SUBAPPLICATION AX_SPLIT_TO_2x_AX_TP (* 1 AX-Eingang gesplittet auf 2 unabhaengig retriggerbare Pulstimer (AX_TP), je eigene Pulsdauer (TQ1/TQ2) und eigener AX-Ausgang (Q1/Q2). Generisch, hardwareunabhaengig. *)
  (* Standard: 61499-2 *)
  (* Version 1.0, 2026-09-09, Franz Höpfinger, Meisterschulen am Ostbahnhof, Ausgelagert aus Uebung_020j2_AX_sub zur Wiederverwendung. *)
  PACKAGE MyLib::sys;
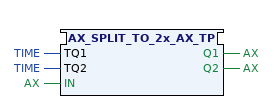
  VAR_INPUT
    TQ1 : TIME;
    TQ2 : TIME;
  END_VAR
  SOCKETS
    IN : adapter::types::unidirectional::AX;
  END_SOCKETS
  PLUGS
    Q1 : adapter::types::unidirectional::AX;
    Q2 : adapter::types::unidirectional::AX;
  END_PLUGS
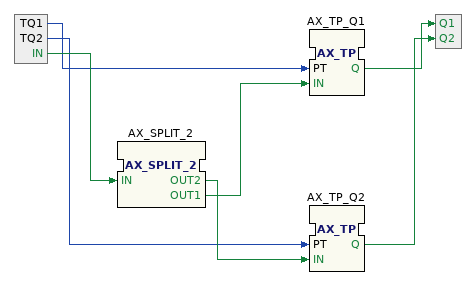
  FBS
    AX_TP_Q2 : adapter::events::unidirectional::timers::AX_TP;
    AX_TP_Q1 : adapter::events::unidirectional::timers::AX_TP;
    AX_SPLIT_2 : adapter::events::unidirectional::AX_SPLIT_2;
  END_FBS
  DATA_CONNECTIONS
    TQ1 TO AX_TP_Q1.PT;
    TQ2 TO AX_TP_Q2.PT;
  END_CONNECTIONS
  ADAPTER_CONNECTIONS
    AX_SPLIT_2.OUT2 TO AX_TP_Q2.IN;
    AX_SPLIT_2.OUT1 TO AX_TP_Q1.IN;
    IN TO AX_SPLIT_2.IN;
    AX_TP_Q2.Q TO Q2;
    AX_TP_Q1.Q TO Q1;
  END_CONNECTIONS
END_SUBAPPLICATION
